FUNCTION_BLOCK FB_ADD_REAL (* REAL Addition *)
  (* Standard: 61499-1-D.1; Classification: Math *)
  (* Version 0.2, 2001-08-05, JHC, Rockwell Automation, Simplified: float add does not throw ArithmeticException. *)
  (* Version 0.1, 2001-04-27, JHC, Rockwell Automation, XML version *)
  (* Version 0.0, 1997-09-13, JHC, Rockwell Automation, SRC version *)
  (* Compiler header: package fb.rt.math; *)
  (* Compiler classdef: class FB_ADD_REAL extends FBFunction2 *)
  (* Compiler Java IBM VisualAge 3.0 *)
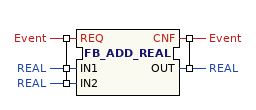
  EVENT_INPUT
    REQ WITH IN1, IN2;
  END_EVENT
  EVENT_OUTPUT
    CNF WITH OUT;
  END_EVENT
  VAR_INPUT
    IN1 : REAL; (* Augend *)
    IN2 : REAL; (* Addend *)
  END_VAR
  VAR_OUTPUT
    OUT : REAL; (* Sum *)
  END_VAR
END_FUNCTION_BLOCK
